FUNCTION_BLOCK dummy (* does nothing *)
  (* Standard: 61499-2 *)
  (* Version 1.0, 2025-12-19, franz *)
  PACKAGE OSCAT::Building::POUs;
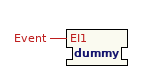
  EVENT_INPUT
    EI1;
  END_EVENT
  EC_STATES
    EI1 : EI1;
  END_STATES
  ALGORITHM EI1 IN ST:

  END_ALGORITHM
END_FUNCTION_BLOCK
